// TIA Portal V18 export
DATA_BLOCK "02_COM"   // DB4, F_DB
{ S7_Optimized_Access := 'TRUE'; DB_Accessible_From_OPC_UA := 'FALSE' }
// stored: DBAccessibleFromOPCUA false
   VAR
      AlwaysFALSE : Bool;
      AlwaysTRUE : Bool := TRUE;
      "!!ITERATOR_STRINGS$$" : Bool;
      "!!02_COM.{matrix_area} FDB$$" { ExternalWritable := 'False'} : Bool;
      "!!02_COM.{matrix_area} PB$$" { ExternalWritable := 'False'} : Bool;
      "!!02_COM.{db_element}$$" { ExternalWritable := 'False'} : Bool;
   END_VAR
BEGIN
END_DATA_BLOCK
